(* CoDeSys 2.3 export: SOC_SIMULATED_TO_VOLTAGE_OUT.EXP *)

(* POU SOC_simulated_to_Voltage_Out, ST *)
PROGRAM SOC_simulated_to_Voltage_Out
VAR
	TheBattery_SOC_simulated: REAL;
	Mixer1_control_signal: REAL;
END_VAR
Mixer1_control_signal := TheBattery_SOC_simulated/10;
END_PROGRAM
